TYPE ACRMemoryIntEvents :
STRUCT
	_Values : ARRAY [0..GCL.cMemoryEventsMAX] OF ACRMemoryIntEvent;
END_STRUCT
END_TYPE

(* stored: Version 1.1.0.1, ProductVersion 3.1.4020.12
   DUT ACRMemoryIntEvents: Id {13f8d2e8-77e6-45f8-9dc0-59e4482daf0a} *)
